INTERFACE I_AssertionMessageList

METHOD AddMessage : BOOL
VAR_INPUT
    Message : T_MaxString;
END_VAR
END_METHOD

METHOD Clear
VAR_INPUT
END_VAR
END_METHOD

END_INTERFACE

(* stored: Version 1.1.0.1, ProductVersion 3.1.4024.4
   Itf I_AssertionMessageList: Id {270b47cc-0623-4afb-ba23-90db3cde0906}
   Method AddMessage: Id {4e3dc3a3-3f3a-4e0a-b8b3-2216c3be2665}
   Method Clear: Id {d5c2c172-7436-4b3f-b473-a575a70ac25f} *)
